FUNCTION_BLOCK EL2819
VAR
	{attribute addProperty Name "WcState"}
	_wcState : WcStateInputToggle;
	{attribute addProperty Name "Info data"}
	_infoData : InfoDataAds;
	_io : EL2819_Data;
END_VAR

PROPERTY IO : REFERENCE TO EL2819_Data
GET
IO REF= _io;
END_GET
END_PROPERTY

PROPERTY WcState : REFERENCE TO WcStateInputToggle
GET
WcState REF= _wcState;
END_GET
END_PROPERTY

END_FUNCTION_BLOCK

(* stored: Version 1.1.0.1, ProductVersion 3.1.4024.9
   POU EL2819: Id {f59ad031-df69-0dad-3dc7-bd4977e4bd0a}, SpecialFunc None
   Property IO: Id {1cfe1976-74d7-0229-2b9b-79837d9d1d6d}
   Get Get: Id {b3e15092-72fc-05c9-1e8a-1747390738f5}
   Property WcState: Id {f8a26ab3-1d06-0816-34c0-3e40777fd7e2}
   Get Get: Id {25ab493c-172e-040d-1d16-e946f9a90b60} *)
